# EPICS autosave request: GalilSup/Db/GALIL_controller_positions.req
$(P)MTR$(CCP)01.DVAL
$(P)MTR$(CCP)02.DVAL
$(P)MTR$(CCP)03.DVAL
$(P)MTR$(CCP)04.DVAL
$(P)MTR$(CCP)05.DVAL
$(P)MTR$(CCP)06.DVAL
$(P)MTR$(CCP)07.DVAL
$(P)MTR$(CCP)08.DVAL
